{attribute 'GeneratedUsingTerminal: EJ7334-0008-0016'}
{attribute addProperty BoxType "EJ7334-0008-0016"}
{attribute addProperty Id "EtcSlaveTerminalBaseDCM_Status_Channel_1AT %I*DCM_Status_Channel_45521CDC8DCM_Status_Channel_2AT %I*DCM_Status_Channel_45521CDC8DCM_Status_Channel_3AT %I*DCM_Status_Channel_45521CDC8DCM_Status_Channel_4AT %I*DCM_Status_Channel_45521CDC8DCM_Outputs_Channel_1AT %Q*DCM_Outputs_Channel_F77F51CE4DCM_Outputs_Channel_2AT %Q*DCM_Outputs_Channel_F77F51CE4DCM_Outputs_Channel_3AT %Q*DCM_Outputs_Channel_F77F51CE4DCM_Outputs_Channel_4AT %Q*DCM_Outputs_Channel_F77F51CE4WcStateAT %I*WcState_9091E0EB2InfoDataAT %I*InfoData_32EB74EA10"}
{attribute addProperty CRC "1839170968"}
{attribute addProperty Size "60"}
TYPE EJ7334_6D9F8598 EXTENDS EtcSlaveTerminalBase :
STRUCT
	{attribute addProperty Name "DCM_Status_Channel_1"}
	DCM_Status_Channel_1 : DCM_Status_Channel_45521CDC;
	{attribute addProperty Name "DCM_Status_Channel_2"}
	DCM_Status_Channel_2 : DCM_Status_Channel_45521CDC;
	{attribute addProperty Name "DCM_Status_Channel_3"}
	DCM_Status_Channel_3 : DCM_Status_Channel_45521CDC;
	{attribute addProperty Name "DCM_Status_Channel_4"}
	DCM_Status_Channel_4 : DCM_Status_Channel_45521CDC;
	{attribute addProperty Name "DCM_Outputs_Channel_1"}
	DCM_Outputs_Channel_1 : DCM_Outputs_Channel_F77F51CE;
	{attribute addProperty Name "DCM_Outputs_Channel_2"}
	DCM_Outputs_Channel_2 : DCM_Outputs_Channel_F77F51CE;
	{attribute addProperty Name "DCM_Outputs_Channel_3"}
	DCM_Outputs_Channel_3 : DCM_Outputs_Channel_F77F51CE;
	{attribute addProperty Name "DCM_Outputs_Channel_4"}
	DCM_Outputs_Channel_4 : DCM_Outputs_Channel_F77F51CE;
	{attribute addProperty Name "WcState"}
	WcState : WcState_9091E0EB;
	{attribute addProperty Name "InfoData"}
	InfoData : InfoData_32EB74EA;
END_STRUCT
END_TYPE

(* stored: Version 1.2.0.0, ProductVersion 3.1.4024.9
   DUT EJ7334_6D9F8598: Id {c4c0938c-39be-47f0-8607-0bae611a7e26} *)
